Staubli VAL3: ROBERT_TP6.dtx

mdesc mRapide100On
mdesc mUsinage20Off = {vel=20, blend=off}
jointRx jStart = {j1=-13.1554864532824, j2=52.8057266959055, j3=128.56179776802, j4=166.840895901009, j5=91.3316286241402, j6=-180.311296989427}
tool tBroche = {x=169.400168374358, y=5.67105066906493E-05, z=47.7499999146672, ry=90, rz=90, fatherId=flange[0], ioLink=valve1}
num nDiametreFraise = 10
frame fPiece = {x=527.606812, y=-37.435701, z=-438.0625, rx=180, rz=-90, fatherId=world[0]}
pointRx pStartUsinage = {x=25, y=25, fatherId=fPiece[0]}
jointRx jChangeOutil = {j1=-4.70104777967739, j2=85.6578357974361, j3=60.0632848818122, j4=174.316678572801, j5=55.8523989241203, j6=-80.7639740285582}
trsf trAppro = {z=-22}
num nPasseRadiale
mdesc mUsinage5Off = {vel=5, blend=off}
